{attribute addProperty BoxType "EK1101-0000-0016"}
{attribute addProperty Id "IDAT %I*UINT162"}
{attribute addProperty CRC "2432610056"}
{attribute addProperty SizeInBites "16"}
{attribute addProperty SizeInBytes "2"}
TYPE ID_90FEAF08 :
STRUCT
	{attribute addProperty Name "ID"}
	ID AT %I* : UINT;
END_STRUCT
END_TYPE

(* stored: Version 1.2.0.0, ProductVersion 3.1.4024.9
   DUT ID_90FEAF08: Id {79adf8f4-09e4-4e9a-8d8c-984ef8be54cb} *)
